PROGRAM Read_Pressure
VAR
	Pressure_Val	: REAL := 0;
	Pressure_Cyl	: REAL := 0;
	
	Hyd_Efficiency	: REAL := 0;
	nBit_Val AT %I*	: UINT;
	nBit_Cyl AT %I*	: UINT;
END_VAR

(* convert to pressure *)
Pressure_Val := (nBit_Val/32767)*160;
Pressure_Cyl := (nBit_Cyl/32767)*160;

(* calculate hyd efficiency *)
//rHyd_Efficiency := Read_Pressure.Pressure_Cyl / Read_Pressure.Pressure_Val;

END_PROGRAM

(* stored: Version 1.1.0.1, ProductVersion 3.1.4024.6
   POU Read_Pressure: Id {4da627ee-194f-436f-bf88-e2e5c518b461}, SpecialFunc None *)
